// TIA Portal V18 export
TYPE "LogInOut_ShW"
// stored: IsFailsafeCompliant false
   STRUCT
      Trigger : Bool;
      OperatorNo : String[48];
      Result : Int;
      Completed : Bool;
   END_STRUCT;
END_TYPE
